Fanuc KAREL source: V_LED_OFF.kl

PROGRAM T
%NOLOCKGROUP
VAR
 v0 : INTEGER
BEGIN
 V_LED_OFF(v0)
END T
